// TIA Portal project "P9" (V17)

(* hardware
DEVICE "S7-1500/ET200MP station_1"  S7-1500 station
   slot 0: "Rail_0"  Rack  6ES7 590-1***0-0AA0
   slot 1: "PLC_1"  CPU 1515-2 PN  6ES7 515-2AM02-0AB0  V2.9
      slot 3: "CPU display_1"  6ES7591-1BA00-0AA0
      slot 32768: "PROFINET interface_1"  X1
         slot 32769: "Port_1"  X1 P1
         slot 32770: "Port_2"  X1 P2
      slot 33024: "PROFINET interface_2"  X2
         slot 33025: "Port_1"  X2 P1
      slot 34817: "Virtual CP interface port_1"  Virtual CP interface port  Virtual CP interface port
*)

// ===== PLC "PLC_1"  CPU 1515-2 PN =====

VAR_GLOBAL   // PLC tag table "Default tag table"
   "START PB" AT %I0.0 : Bool;
   "STOP PB" AT %I0.1 : Bool;
   "EMPTY BOTTLE DETECTION" AT %I0.2 : Bool;
   "BOTTLE DETECTOR" AT %I0.3 : Bool;
   "CYCLE ON" AT %Q0.0 : Bool;
   "CONVEYOR ON" AT %Q0.1 : Bool;
   "CYLINDER ON" AT %Q0.2 : Bool;
   "RELAY COIL" AT %M11.0 : Bool;
   "POSITIVE EDGE" AT %M0.0 : Bool;
   "SWIFT REGISTER" AT %MW10 : Int;
   "SHIFT BIT" AT %M11.5 : Bool;
END_VAR

ORGANIZATION_BLOCK "Main"   // OB1, LAD, ProgramCycle
TITLE = "Main Program Sweep (Cycle)"
{ S7_Optimized_Access := 'TRUE' }
VERSION : 0.1
   VAR_INPUT
      Initial_Call : Bool;   // Initial call of this OB
      Remanence : Bool;   // =True, if remanent data are available
   END_VAR
   VAR_TEMP   // added for the SCL form of the ladder/FBD networks
      _w1 : Bool;
      _w2 : Bool;
   END_VAR
BEGIN

REGION Network 1
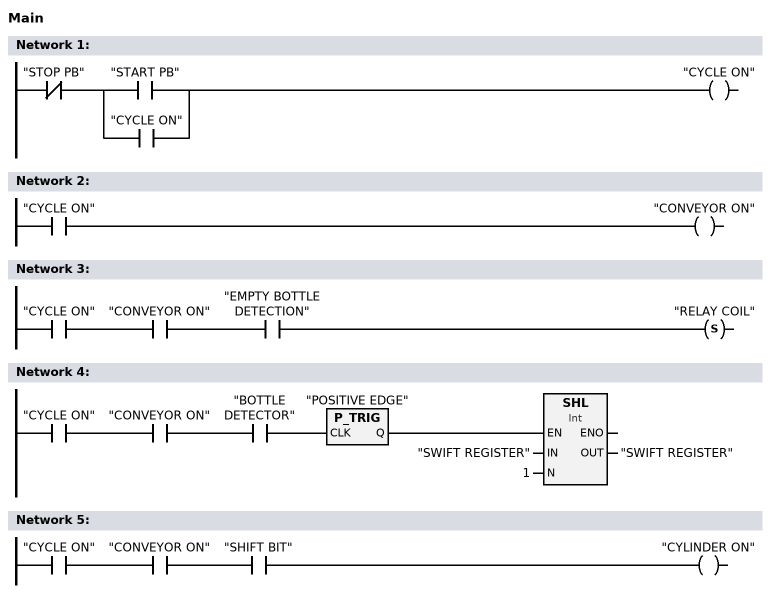
   RUNG wire#powerrail
      I_Contact( "STOP PB" )
      wire#w1
      Contact( "START PB" )
      wire#w2
      Coil( "CYCLE ON" )
   END_RUNG
   RUNG wire#w1
      Contact( "CYCLE ON" )
   END_RUNG wire#w2
   // the same network as SCL:
   "CYCLE ON" := NOT "STOP PB" AND ("START PB" OR "CYCLE ON");
END_REGION

REGION Network 2
   RUNG wire#powerrail
      Contact( "CYCLE ON" )
      Coil( "CONVEYOR ON" )
   END_RUNG
   // the same network as SCL:
   "CONVEYOR ON" := "CYCLE ON";
END_REGION

REGION Network 3
   RUNG wire#powerrail
      Contact( "CYCLE ON" )
      Contact( "CONVEYOR ON" )
      Contact( "EMPTY BOTTLE DETECTION" )
      S_Coil( "RELAY COIL" )
   END_RUNG
   // the same network as SCL:
   IF "CYCLE ON" AND "CONVEYOR ON" AND "EMPTY BOTTLE DETECTION" THEN "RELAY COIL" := TRUE; END_IF;
END_REGION

REGION Network 4
   RUNG wire#powerrail
      Contact( "CYCLE ON" )
      Contact( "CONVEYOR ON" )
      Contact( "BOTTLE DETECTOR" )
      P_Trig( "POSITIVE EDGE" )
      { S7_Templates := "SrcType := Int" } Shl(in := "SWIFT REGISTER", n := 1, out => "SWIFT REGISTER")
   END_RUNG
   // the same network as SCL:
   #_w1 := "CYCLE ON" AND "CONVEYOR ON" AND "BOTTLE DETECTOR";
   #_w2 := #_w1 AND NOT "POSITIVE EDGE";   // rising edge
   "POSITIVE EDGE" := #_w1;
   IF #_w2 THEN "SWIFT REGISTER" := SHL(IN := "SWIFT REGISTER", N := 1); END_IF;
END_REGION

REGION Network 5
   RUNG wire#powerrail
      Contact( "CYCLE ON" )
      Contact( "CONVEYOR ON" )
      Contact( "SHIFT BIT" )
      Coil( "CYLINDER ON" )
   END_RUNG
   // the same network as SCL:
   "CYLINDER ON" := "CYCLE ON" AND "CONVEYOR ON" AND "SHIFT BIT";
END_REGION
END_ORGANIZATION_BLOCK